// Function block for creating custom errors.
{attribute 'enable_dynamic_creation'}
{attribute 'reflection'}
{attribute 'no_explicit_call' := 'direct call for this function block is not allowed'} 
FUNCTION_BLOCK FINAL FsFB_ErrorDefinition EXTENDS FsFB_Error
VAR
END_VAR

PROPERTY Code : FsT_ErrCode
SET
THIS^._Code := Code;
END_SET
END_PROPERTY

PROPERTY PROTECTED DynamicTypeName : FsT_Str
GET
VAR
	fbVar : FsFB_ErrorDefinition;
	VarInfo : FsT_VarInfo := __VARINFO(fbVar); 
END_VAR
DynamicTypeName := VarInfo.TypeName;
END_GET
END_PROPERTY

PROPERTY Message : FsT_ErrSrc
SET
THIS^._Message := Message;
END_SET
END_PROPERTY

END_FUNCTION_BLOCK

(* stored: Version 1.1.0.1, ProductVersion 3.1.4024.4
   POU FsFB_ErrorDefinition: Id {2e34dc7b-c479-4572-b7c4-2d509ca0d2fa}, SpecialFunc None
   Folder Properties: Id {b0caec45-c7ea-4b26-b385-9263908a2397}
   Property Code: Id {ea2cf2a8-f62d-4b13-a982-1df0ca0b8500}
   Set Set: Id {11edbd4e-def0-4198-87f2-c70903214c61}
   Property DynamicTypeName: Id {b277e546-6883-4ab0-8e7b-37beec70524f}
   Get Get: Id {1c94e104-78d3-404c-9dc0-38e7ba841180}
   Property Message: Id {97cc91a0-f032-4444-83bc-ce65a659717b}
   Set Set: Id {4ffc18b8-0c38-41a6-9f1a-2f6a818b00ea} *)
